Xinje XCPPro project, PLC1: XC3-14 (software 3.3r 2017-11-30)

PROGRAM Ladder

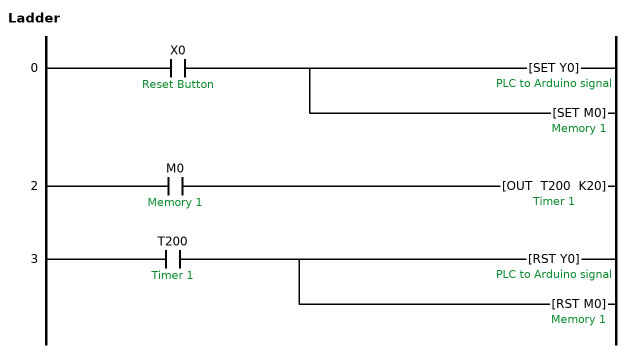
LD     X0	; Reset Button
SET    Y0	; PLC to Arduino signal
SET    M0	; Memory 1
LD     M0	; Memory 1
OUT    T200 K20	; Timer 1
LD     T200	; Timer 1
RST    Y0	; PLC to Arduino signal
RST    M0	; Memory 1